FUNCTION_BLOCK AX_SELECT (* selection between two events based on boolean input G *)
  (* Standard: 61499-1 Annex A; Description: Copyright (c) 2017 fortiss GmbH This program and the accompanying materials are made available under the terms of the Eclipse Public License 2.0 which is available at https://www.eclipse.org/legal/epl-2.0/ SPDX-License-Identifier: EPL-2.0 *)
  (* Version 3.0, 2025-04-14, Patrick Aigner, changed package *)
  (* Version 1.0, 2017-09-21, Alois Zoitl, fortiss GmbH, initial API and implementation and/or initial documentation *)
  PACKAGE adapter::events::unidirectional;
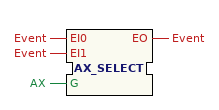
  EVENT_INPUT
    EI0; (* Input event, selected when G=0 *)
    EI1; (* Input event, selected when G=1 *)
  END_EVENT
  EVENT_OUTPUT
    EO; (* Output Event *)
  END_EVENT
  SOCKETS
    G : adapter::types::unidirectional::AX; (* Select EI0 when G=0, EI1 when G=1 *)
  END_SOCKETS
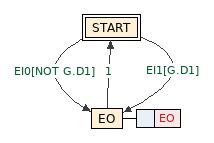
  EC_STATES
    START; (* Initial State *)
    EO : -> EO; (* Issue Output Event *)
  END_STATES
  EC_TRANSITIONS
    EO TO START := 1;
    START TO EO := EI0[NOT G.D1];
    START TO EO := EI1[G.D1];
  END_TRANSITIONS
END_FUNCTION_BLOCK
